SYSTEM TEST_VSTYLE (* Test Display of VSTYLE values *)
  (* Standard: 61499-1 *)
  (* Version 0.0, 2000-05-27, JHC, Rockwell Automation *)
  DEVICE HMI : FRAME_DEVICE
    RESOURCE RES1 : PANEL_RESOURCE
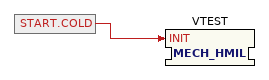
      FBS
        VTEST : MECH_HMIL;
      END_FBS
      EVENT_CONNECTIONS
        START.COLD TO VTEST.INIT;
      END_CONNECTIONS
    END_RESOURCE
  END_DEVICE
  DEVICE VIEW : FRAME_DEVICE
    RESOURCE RES1 : PANEL_RESOURCE
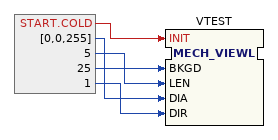
      FBS
        VTEST : MECH_VIEWL;
      END_FBS
      EVENT_CONNECTIONS
        START.COLD TO VTEST.INIT;
      END_CONNECTIONS
      DATA_CONNECTIONS
        [0,0,255] TO VTEST.BKGD;
        5 TO VTEST.LEN;
        25 TO VTEST.DIA;
        1 TO VTEST.DIR;
      END_CONNECTIONS
    END_RESOURCE
  END_DEVICE
  DATA_CONNECTIONS (* parameter values *)
    [100,100,330,80] TO HMI.BOUNDS;
    [430,100,40,175] TO VIEW.BOUNDS;
  END_CONNECTIONS
END_SYSTEM
